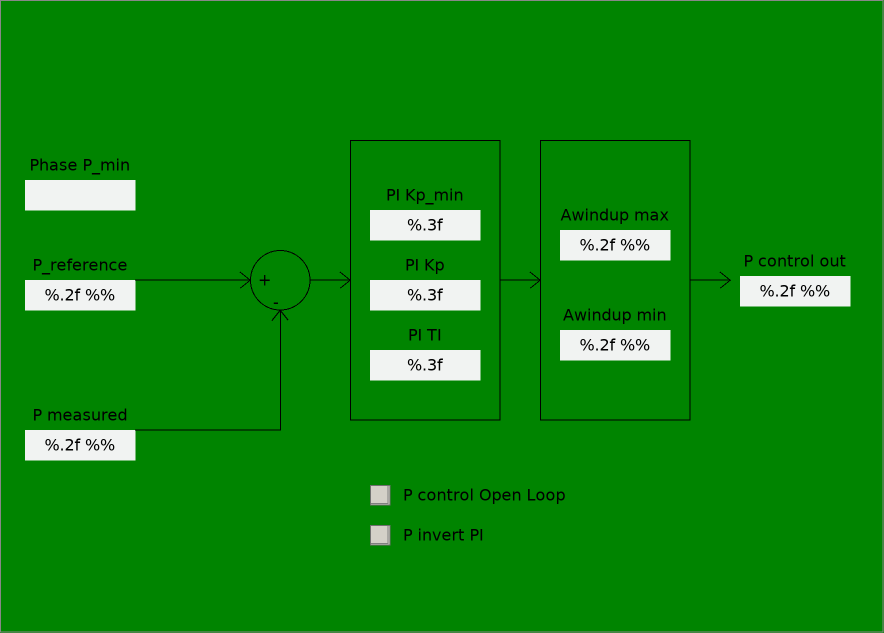
VISUALIZATION P_controller  // 884x633
    Rectangle (540,140 150x280)
    Rectangle (350,140 150x280)
    Rectangle (25,280 110x30), "%.2f %%", text variable: GVL_HANDLER.GUI_vars[P_reference]
        OnMouseDown: write the text variable via Default
    Rectangle (25,250 110x30), "P_reference"
    Rectangle (25,430 110x30), "%.2f %%", text variable: GVL_HANDLER.GUI_vars[P_feedback]
        OnMouseDown: write the text variable via Default
    Rectangle (25,400 110x30), "P measured"
    Line (250,280) (135,280)
    Ellipse (250,250 60x60)
    Line (280,430) (135,430)
    Line (280,310) (280,430)
    Line (288,320) (280,310)
    Line (272,320) (280,310)
    Line (250,280) (240,288)
    Line (250,280) (240,272)
    Line (350,280) (340,288)
    Line (350,280) (310,280)
    Line (350,280) (340,272)
    Rectangle (370,280 110x30), "%.3f", text variable: GVL_HANDLER.GUI_vars[P_kp]
        OnMouseClick: write the text variable via Default
    Rectangle (370,250 110x30), "PI Kp"
    Rectangle (370,350 110x30), "%.3f", text variable: GVL_HANDLER.GUI_vars[P_ti]
        OnMouseClick: write the text variable via Default
    Rectangle (370,320 110x30), "PI TI"
    Rectangle (370,210 110x30), "%.3f", text variable: GVL_HANDLER.GUI_vars[P_kp_min]
        OnMouseClick: write the text variable via Default
    Rectangle (370,180 110x30), "PI Kp_min"
    Line (540,280) (530,288)
    Line (540,280) (500,280)
    Line (540,280) (530,272)
    Rectangle (560,330 110x30), "%.2f %%", text variable: GVL_HANDLER.GUI_vars[P_low]
        OnMouseClick: write the text variable via Default
    Rectangle (560,300 110x30), "Awindup min"
    Rectangle (560,230 110x30), "%.2f %%", text variable: GVL_HANDLER.GUI_vars[P_high]
        OnMouseClick: write the text variable via Default
    Rectangle (560,200 110x30), "Awindup max"
    Line (730,280) (720,288)
    Line (730,280) (690,280)
    Line (730,280) (720,272)
    Rectangle (740,276 110x30), "%.2f %%", text variable: GVL_HANDLER.GUI_vars[P_output]
    Rectangle (740,246 110x30), "P control out"
    Rectangle (400,480 170x30), "P control Open Loop"
    Rectangle (400,520 170x30), "P invert PI"
    Button (370,485 20x20), colour toggle: GVL_GUI.P_OL_sel_button
        OnMouseClick: toggle GVL_HANDLER.GUI_vars[P_loop]
        OnMouseClick: execute {
            IF GVL_GUI.P_OL_sel_button = 0 THEN
            	GVL_GUI.P_OL_sel_button:= 1;
            ELSE
            	GVL_GUI.P_OL_sel_button:= 0;
            END_IF
        }
    Button (370,525 20x20), colour toggle: GVL_GUI.P_invert_button
        OnMouseClick: toggle GVL_HANDLER.GUI_vars[P_invert]
        OnMouseClick: execute {
            IF GVL_GUI.P_invert_button = 0 THEN
            	GVL_GUI.P_invert_button:= 1;
            ELSE
            	GVL_GUI.P_invert_button:= 0;
            END_IF
        }
    Rectangle (255,265 110x30), "+"
    Rectangle (270,287 110x30), "-"
    Rectangle (25,180 110x30), text list: 'P_min_indicator', text index: GVL_POWERMETER.P_min_indicator
    Rectangle (25,150 110x30), "Phase P_min"
END_VISUALIZATION

(* stored: Version 1.1.0.1, ProductVersion 3.1.4024.11
   Visu P_controller: Id {fdf8bad8-7dec-4e99-87e6-24546c589c9b} *)
